// TwinCAT 3 PLC project Main
// ProgramVersion: 3.1.4023.0
// libraries:
//   Tc2_Standard, * (Beckhoff Automation GmbH)
//   Tc2_System, * (Beckhoff Automation GmbH)
//   Tc3_Module, * (Beckhoff Automation GmbH)
// project tree:
//   DUTs/ MySecondStructure.TcDUT, MyStructure.TcDUT
//   / PlcTask.TcTTO
//   POUs/ MAIN.TcPOU
// real-time tasks:
//   TASK PlcTask: cycle T#10ms, priority 20, ADS port 350

CONFIGURATION Main
    RESOURCE PLC ON TwinCAT3
        TASK PlcTask(INTERVAL := T#10ms, PRIORITY := 20);
        PROGRAM MAIN WITH PlcTask : MAIN;
    END_RESOURCE
END_CONFIGURATION

// ---- DUTs/MySecondStructure.TcDUT
TYPE MySecondStructure :
STRUCT
	myLint : LINT;
	myDint : DINT;
END_STRUCT
END_TYPE

// ---- DUTs/MyStructure.TcDUT
TYPE MyStructure :
STRUCT
	myBool : BOOL;
	myArrayOfBool : ARRAY [0..10] OF BOOL;
	myReal : REAL;
	myArrayOfStructures : ARRAY [0..1] OF MySecondStructure;
END_STRUCT
END_TYPE

// ---- POUs/MAIN.TcPOU
PROGRAM MAIN
VAR
	initalized : BOOL;
	pMyArrayOfStructures : POINTER TO ARRAY [0..2] OF MyStructure;

END_VAR

IF NOT initalized THEN
	
	pMyArrayOfStructures := __NEW(BYTE, SIZEOF(ARRAY [0..2] OF MyStructure));
	initalized := TRUE;
	
END_IF
pMyArrayOfStructures^[2].myBool := true;
pMyArrayOfStructures^[2].myArrayOfBool[2] := TRUE;
pMyArrayOfStructures^[2].myArrayOfStructures[1].myDint := 123;
pMyArrayOfStructures^[2].myReal := 3.142;

END_PROGRAM
